FUNCTION_BLOCK SS5a_Camera (* Basic FB with empty ECC *)
  (* Standard: 61499-2 *)
  (* Version 1.0, 2024-10-03, DEVIASH *)
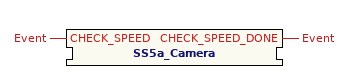
  EVENT_INPUT
    CHECK_SPEED;
  END_EVENT
  EVENT_OUTPUT
    CHECK_SPEED_DONE;
  END_EVENT
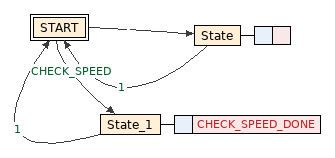
  EC_STATES
    START; (* Initial State *)
    State;
    State_1 : -> CHECK_SPEED_DONE;
  END_STATES
  EC_TRANSITIONS
    START TO State := ;
    State TO START := 1;
    START TO State_1 := CHECK_SPEED;
    State_1 TO START := 1;
  END_TRANSITIONS
END_FUNCTION_BLOCK
